FUNCTION_BLOCK PUBLIC FB_LampOnOff
VAR
	nLightLevel			: USINT;
END_VAR

// Reduces the control value by 5 in the range of 10 to 100.
METHOD PUBLIC DimDown
Off();
END_METHOD

// Increments the control value by 5 in the range of 10 to 100.
METHOD PUBLIC DimUp
On();
END_METHOD

// Sets the control value to 0.
METHOD PUBLIC Off
nLightLevel := 0;
END_METHOD

// Sets the control value to 100.
METHOD PUBLIC On
nLightLevel := 100;
END_METHOD

END_FUNCTION_BLOCK

(* stored: Version 1.1.0.1, ProductVersion 3.1.4024.12
   POU FB_LampOnOff: Id {55e66dc1-05c3-43f8-9bc8-5075ca0cd865}, SpecialFunc None
   Method DimDown: Id {561a1d70-9f10-40d7-ba32-1dcaaac84037}
   Method DimUp: Id {7736046e-8f67-492e-b22e-d97f488e1604}
   Method Off: Id {54f23483-66d0-4707-9581-54558ff84187}
   Method On: Id {ea9cd1d9-8590-4b0b-b6ec-c19fb0ca1b1d} *)
